# EPICS StreamDevice protocol: iocs/serialKistlerOld/iocBoot/protocols/quantel.proto
## Quantel Protocol file
#Terminator = CR LF;
#Terminator =CR; does not work
#Terminator =LF; # OK
# CTRL+J (<LF>)  \n
OutTerminator = LF; # OK
#messages have always "\r\n" plus 15 chars
MaxInput = 17;
######################
getVoltage {
    out "V"; in "\r\nvoltage %u V";
}

setTrigger {
    out "Q%2d%(\$1)2d%(\$2)2d";
    @init { out "Q"; in "\r\nQS  %2d  %(\$1)2d  %(\$2)2d";}
}

getTrigger {
    out "Q";
    in "\r\nQS  %2d  %(\$1)2d  %(\$2)2d";
}

setStandby{
    out "S";
}
#
getMode{
    out "";
    in  "\r\n%{standby        |simmer         |fire auto      }"
}
setMode{
    out "%{S|M|A|CC}";
    in  "\r\n%{standby        |simmer         |fire auto      |fire auto      }"
}

# Connect a stringout record to this to get
# a generic command interface.
# After processing finishes, the record contains the reply.

debug {
    ExtraInput = Ignore;
    out "%s"; in "%39c"

}
